{attribute addProperty BoxType "EJ2918-0000-0017"}
{attribute addProperty Id "Module_1_FSOEModule_1_FSOE_FC73D945104130Module_2_FSOUTModule_2_FSOUT_15E085466480Module_3_DEVICEIOModule_3_DEVICEIO_FB2B67D71620Module_4_FSLOGICModule_4_FSLOGIC_3E6251391620WcStateAT %I*WcState_DC9C971540.50InfoDataAT %I*InfoData_BC63D37F80100"}
{attribute addProperty CRC "2831312890"}
{attribute addProperty SizeInBites "284"}
{attribute addProperty SizeInBytes "35.5"}
TYPE EJ2918_AA36864B :
STRUCT
	{attribute addProperty Name "Module_1_FSOE"}
	Module_1_FSOE : Module_1_FSOE_FC73D945;
	{attribute addProperty Name "Module_2_FSOUT"}
	Module_2_FSOUT : Module_2_FSOUT_15E08546;
	{attribute addProperty Name "Module_3_DEVICEIO"}
	Module_3_DEVICEIO : Module_3_DEVICEIO_FB2B67D7;
	{attribute addProperty Name "Module_4_FSLOGIC"}
	Module_4_FSLOGIC : Module_4_FSLOGIC_3E625139;
	{attribute addProperty Name "WcState"}
	WcState : WcState_DC9C9715;
	{attribute addProperty Name "InfoData"}
	InfoData : InfoData_BC63D37F;
END_STRUCT
END_TYPE

(* stored: Version 1.2.0.0, ProductVersion 3.1.4024.9
   DUT EJ2918_AA36864B: Id {3a721550-9081-476b-8062-0baad5e09b71} *)
